FUNCTION F_NcErrorMessage : STRING[2048]
VAR_INPUT
	Error		: UDINT;
END_VAR

CASE Error OF
		0		: 		F_NcErrorMessage	:= 'None';

(* --> User defined errors for entire machine <--*)
		1		:		F_NcErrorMessage	:= 'The machine is in error at startup - please reset. ';		

		ELSE
			IF 36844 < Error AND Error < 36857 THEN
				F_NcErrorMessage:='NC3_Internal_Unexpected INTERNAL Error';
			ELSE		
				F_NcErrorMessage:='Msg Unknown';
			END_IF	

END_CASE

END_FUNCTION

(* stored: Version 1.1.0.1, ProductVersion 3.1.4024.9
   POU F_NcErrorMessage: Id {c6550364-7eba-4899-8a2d-15b3499de212}, SpecialFunc None *)
